// TIA Portal V20 export
DATA_BLOCK "Config"   // DB67
{ DB_Accessible_From_OPC_UA := 'FALSE' }
AUTHOR : ERsystem_FA2_DH. Kim
// stored: Access Published, DBAccessibleFromOPCUA false, DBAccessibleFromWebserver false, MemoryReserve 100, Namespace Unit1.Em3
   VAR RETAIN
      em { ExternalWritable := 'False'} : "LAF_typeEmConfiguration";
      axis { ExternalAccessible := 'False'; ExternalVisible := 'False'; ExternalWritable := 'False'} : Array[1.._.U1EM3_NO_OF_AXES] of DB_ANY;
      cam : Array[1.._.U1EM3_NO_OF_CAM] of DB_ANY;
      cmSafetyPinIdlePositionSensor { S7_SetPoint := 'True'} : "LBC_typeDigitalSignalConfiguration";
      cmRotationSafetyPinPositionSensor { S7_SetPoint := 'True'} : "LBC_typeDigitalSignalConfiguration";
      cmIonizerTopMaintDetection { S7_SetPoint := 'True'} : "LBC_typeDigitalSignalConfiguration";
      cmIonizerTopErrorDetection { S7_SetPoint := 'True'} : "LBC_typeDigitalSignalConfiguration";
      cmIonizerBtmMaintDetection { S7_SetPoint := 'True'} : "LBC_typeDigitalSignalConfiguration";
      cmIonizerBtmErrorDetection { S7_SetPoint := 'True'} : "LBC_typeDigitalSignalConfiguration";
      cmDancerEncoder { ExternalAccessible := 'False'; ExternalVisible := 'False'; ExternalWritable := 'False'} : "LBC_typeAnalogInputConfiguration";
      cmDancerElectroPneumaticRegulator { ExternalAccessible := 'False'; ExternalVisible := 'False'; ExternalWritable := 'False'} : "LBC_typeAnalogOutputConfiguration";
      cmCompensatorAxisX { ExternalAccessible := 'False'; ExternalVisible := 'False'; ExternalWritable := 'False'} : "LBC_typeAxis64PosConfiguration";
      cmMasterVirtualAxis { S7_SetPoint := 'True'} : "LBC_typeAxis64PosConfiguration";
      cmUnwinderVirtualAxis : "LBC_typeAxis64PosConfiguration";
      cmDancerFwdBwd { ExternalAccessible := 'False'; ExternalVisible := 'False'; ExternalWritable := 'False'} : "LBC_typeTwoWayActuatorConfiguration";
      cmSepaUnwinderIonizerTop { ExternalAccessible := 'False'; ExternalVisible := 'False'; ExternalWritable := 'False'; S7_SetPoint := 'True'} : "LBC_typeTwoWayActuatorConfiguration";
      cmSepaUnwinderIonizerBottom { ExternalAccessible := 'False'; ExternalVisible := 'False'; ExternalWritable := 'False'; S7_SetPoint := 'True'} : "LBC_typeTwoWayActuatorConfiguration";
      cmEpcPivot { ExternalAccessible := 'False'; ExternalVisible := 'False'; ExternalWritable := 'False'} : "LER_typeCON600Configuration";
      cmLoadCellControllerInterface { ExternalAccessible := 'False'; ExternalVisible := 'False'; ExternalWritable := 'False'} : "LBC_typeAnalogInputConfiguration";
      softCam : Struct
         cmCompensatorAxisX : "LER_typeSoftCamInterface";
         cmMasterVirtualAxis { S7_SetPoint := 'True'} : "LER_typeSoftCamInterface";
         cmUnwinderVirtualAxis { S7_SetPoint := 'True'} : "LER_typeSoftCamInterface";
      END_STRUCT;
   END_VAR
BEGIN
   em.referenceDesignator.parent := WSTRING#'U1';
   em.referenceDesignator.relative := WSTRING#'EM3 WebGuide';
   em.referenceDesignator.combined := WSTRING#'U1.EM3 WebGuide';
   axis[1] := 85;   // BA030AZSDR3_CompensatorAxisX
   axis[2] := 117;   // BA030A_MasterAxis
   axis[3] := 143;   // BA030A_UnwinderVirtualAxis
   cam[1] := 69;   // BA030AZSDR3_CompensatorAxisX_Cam
   cam[2] := 73;   // BA030AZSDR4_SepaFeedingRollerAxisB_Cam
   cmSafetyPinIdlePositionSensor.referenceDesignator := WSTRING#'DigitalSignal';
   cmSafetyPinIdlePositionSensor.onDelay := T#0MS;
   cmSafetyPinIdlePositionSensor.offDelay := T#0MS;
   cmSafetyPinIdlePositionSensor.default := FALSE;
   cmSafetyPinIdlePositionSensor.invertProcessValue := FALSE;
   cmSafetyPinIdlePositionSensor.disableAlarms := FALSE;
   cmRotationSafetyPinPositionSensor.referenceDesignator := WSTRING#'DigitalSignal';
   cmRotationSafetyPinPositionSensor.onDelay := T#0MS;
   cmRotationSafetyPinPositionSensor.offDelay := T#0MS;
   cmRotationSafetyPinPositionSensor.default := FALSE;
   cmRotationSafetyPinPositionSensor.invertProcessValue := FALSE;
   cmRotationSafetyPinPositionSensor.disableAlarms := FALSE;
   cmIonizerTopMaintDetection.referenceDesignator := WSTRING#'DigitalSignal';
   cmIonizerTopMaintDetection.onDelay := T#0MS;
   cmIonizerTopMaintDetection.offDelay := T#0MS;
   cmIonizerTopMaintDetection.default := FALSE;
   cmIonizerTopMaintDetection.invertProcessValue := FALSE;
   cmIonizerTopMaintDetection.disableAlarms := FALSE;
   cmIonizerTopErrorDetection.referenceDesignator := WSTRING#'DigitalSignal';
   cmIonizerTopErrorDetection.onDelay := T#0MS;
   cmIonizerTopErrorDetection.offDelay := T#0MS;
   cmIonizerTopErrorDetection.default := FALSE;
   cmIonizerTopErrorDetection.invertProcessValue := FALSE;
   cmIonizerTopErrorDetection.disableAlarms := FALSE;
   cmIonizerBtmMaintDetection.referenceDesignator := WSTRING#'DigitalSignal';
   cmIonizerBtmMaintDetection.onDelay := T#0MS;
   cmIonizerBtmMaintDetection.offDelay := T#0MS;
   cmIonizerBtmMaintDetection.default := FALSE;
   cmIonizerBtmMaintDetection.invertProcessValue := FALSE;
   cmIonizerBtmMaintDetection.disableAlarms := FALSE;
   cmIonizerBtmErrorDetection.referenceDesignator := WSTRING#'DigitalSignal';
   cmIonizerBtmErrorDetection.onDelay := T#0MS;
   cmIonizerBtmErrorDetection.offDelay := T#0MS;
   cmIonizerBtmErrorDetection.default := FALSE;
   cmIonizerBtmErrorDetection.invertProcessValue := FALSE;
   cmIonizerBtmErrorDetection.disableAlarms := FALSE;
   cmDancerEncoder.referenceDesignator := WSTRING#'cmDancerEncoder';
   cmDancerEncoder.physicalUnit := 'unit';
   cmDancerEncoder.isUnipolarSignal := TRUE;
   cmDancerEncoder.default := 0.0;
   cmDancerEncoder.limitHigh2 := 20.0;
   cmDancerEncoder.limitHigh1 := 15.0;
   cmDancerEncoder.limitLow1 := -15.0;
   cmDancerEncoder.limitLow2 := -50.0;
   cmDancerEncoder.processValueMax := 43.0;
   cmDancerEncoder.processValueMin := -43.0;
   cmDancerEncoder.scaleAnalogUppPoint := 27648.0;
   cmDancerEncoder.scaleAnalogLowPoint := 0.0;
   cmDancerEncoder.scaleProcessUppPoint := 43.0;
   cmDancerEncoder.scaleProcessLowPoint := -43.0;
   cmDancerEncoder.disableAlarms := FALSE;
   cmDancerElectroPneumaticRegulator.referenceDesignator := WSTRING#'cmDancerRegulator';
   cmDancerElectroPneumaticRegulator.physicalUnit := 'unit';
   cmDancerElectroPneumaticRegulator.isUnipolarSignal := TRUE;
   cmDancerElectroPneumaticRegulator.default := 0;
   cmDancerElectroPneumaticRegulator.limitHigh2 := 0.5;
   cmDancerElectroPneumaticRegulator.limitHigh1 := 0.5;
   cmDancerElectroPneumaticRegulator.limitLow1 := 0.0;
   cmDancerElectroPneumaticRegulator.limitLow2 := 0.0;
   cmDancerElectroPneumaticRegulator.processValueMax := 0.5;
   cmDancerElectroPneumaticRegulator.processValueMin := 0.0;
   cmDancerElectroPneumaticRegulator.scaleProcessUppPoint := 0.5;
   cmDancerElectroPneumaticRegulator.scaleProcessLowPoint := 0.0;
   cmDancerElectroPneumaticRegulator.scaleAnalogUppPoint := 27648.0;
   cmDancerElectroPneumaticRegulator.scaleAnalogLowPoint := 0.0;
   cmDancerElectroPneumaticRegulator.disableAlarms := TRUE;
   cmCompensatorAxisX.referenceDesignator := WSTRING#'cmCompensatorAxisX';
   cmCompensatorAxisX.disableAlarms := FALSE;
   cmCompensatorAxisX.masterControlPopUp := TRUE;
   cmCompensatorAxisX.setPositions[0].position := 0.0;
   cmCompensatorAxisX.setPositions[1].position := 50.0;
   cmCompensatorAxisX.setPositions[2].position := 70.0;
   cmCompensatorAxisX.setPositions[3..15].position := 0.0;
   cmCompensatorAxisX.setPositions[0].velocity := -1.0;
   cmCompensatorAxisX.setPositions[1..2].velocity := 30.0;
   cmCompensatorAxisX.setPositions[3..15].velocity := -1.0;
   cmCompensatorAxisX.setPositions[0].acceleration := -1.0;
   cmCompensatorAxisX.setPositions[1..2].acceleration := 30.0;
   cmCompensatorAxisX.setPositions[3..15].acceleration := -1.0;
   cmCompensatorAxisX.setPositions[0].deceleration := -1.0;
   cmCompensatorAxisX.setPositions[1..2].deceleration := 30.0;
   cmCompensatorAxisX.setPositions[3..15].deceleration := -1.0;
   cmCompensatorAxisX.setPositions[0..15]."name" := '';
   cmUnwinderVirtualAxis.referenceDesignator := WSTRING#'Axis64Pos';
   cmUnwinderVirtualAxis.disableAlarms := TRUE;
   cmUnwinderVirtualAxis.masterControlPopUp := TRUE;
   cmUnwinderVirtualAxis.setPositions[0..15].position := 0.0;
   cmUnwinderVirtualAxis.setPositions[0..15].velocity := -1.0;
   cmUnwinderVirtualAxis.setPositions[0..15].acceleration := -1.0;
   cmUnwinderVirtualAxis.setPositions[0..15].deceleration := -1.0;
   cmUnwinderVirtualAxis.setPositions[0..15]."name" := '';
   cmDancerFwdBwd.referenceDesignator := WSTRING#'cmDancerFwdBwd';
   cmDancerFwdBwd.monitoringLeavingFeedback := T#1S;
   cmDancerFwdBwd.monitoringReachingFeedback := T#1S;
   cmDancerFwdBwd.monitoringDiscrepancy := T#0MS;
   cmDancerFwdBwd.setOutputHomeContinuously := TRUE;
   cmDancerFwdBwd.setOutputWorkContinuously := TRUE;
   cmDancerFwdBwd.disableHomeCommand := FALSE;
   cmDancerFwdBwd.disableFeedbackHomePos := TRUE;
   cmDancerFwdBwd.disableFeedbackWorkPos := TRUE;
   cmDancerFwdBwd.disableAlarms := TRUE;
   cmDancerFwdBwd.resetOutputsOnError := FALSE;
   cmDancerFwdBwd.allwaysWaitOnReachingTime := FALSE;
   cmSepaUnwinderIonizerTop.referenceDesignator := WSTRING#'cmSepaUnwinderIonizerTop';
   cmSepaUnwinderIonizerTop.monitoringLeavingFeedback := T#500ms;
   cmSepaUnwinderIonizerTop.monitoringReachingFeedback := T#500ms;
   cmSepaUnwinderIonizerTop.monitoringDiscrepancy := T#0MS;
   cmSepaUnwinderIonizerTop.setOutputHomeContinuously := TRUE;
   cmSepaUnwinderIonizerTop.setOutputWorkContinuously := TRUE;
   cmSepaUnwinderIonizerTop.disableHomeCommand := FALSE;
   cmSepaUnwinderIonizerTop.disableFeedbackHomePos := TRUE;
   cmSepaUnwinderIonizerTop.disableFeedbackWorkPos := TRUE;
   cmSepaUnwinderIonizerTop.disableAlarms := TRUE;
   cmSepaUnwinderIonizerTop.resetOutputsOnError := FALSE;
   cmSepaUnwinderIonizerTop.allwaysWaitOnReachingTime := FALSE;
   cmSepaUnwinderIonizerBottom.referenceDesignator := WSTRING#'cmSepaUnwinderIonizerBtm';
   cmSepaUnwinderIonizerBottom.monitoringLeavingFeedback := T#500ms;
   cmSepaUnwinderIonizerBottom.monitoringReachingFeedback := T#500ms;
   cmSepaUnwinderIonizerBottom.monitoringDiscrepancy := T#0MS;
   cmSepaUnwinderIonizerBottom.setOutputHomeContinuously := TRUE;
   cmSepaUnwinderIonizerBottom.setOutputWorkContinuously := TRUE;
   cmSepaUnwinderIonizerBottom.disableHomeCommand := FALSE;
   cmSepaUnwinderIonizerBottom.disableFeedbackHomePos := TRUE;
   cmSepaUnwinderIonizerBottom.disableFeedbackWorkPos := TRUE;
   cmSepaUnwinderIonizerBottom.disableAlarms := TRUE;
   cmSepaUnwinderIonizerBottom.resetOutputsOnError := FALSE;
   cmSepaUnwinderIonizerBottom.allwaysWaitOnReachingTime := FALSE;
   cmLoadCellControllerInterface.referenceDesignator := WSTRING#'cmLoadCellController';
   cmLoadCellControllerInterface.physicalUnit := 'unit';
   cmLoadCellControllerInterface.isUnipolarSignal := TRUE;
   cmLoadCellControllerInterface.default := 0.0;
   cmLoadCellControllerInterface.limitHigh2 := 90.0;
   cmLoadCellControllerInterface.limitHigh1 := 80.0;
   cmLoadCellControllerInterface.limitLow1 := -80.0;
   cmLoadCellControllerInterface.limitLow2 := -90.0;
   cmLoadCellControllerInterface.processValueMax := 100.0;
   cmLoadCellControllerInterface.processValueMin := -100.0;
   cmLoadCellControllerInterface.scaleAnalogUppPoint := 27648.0;
   cmLoadCellControllerInterface.scaleAnalogLowPoint := 0.0;
   cmLoadCellControllerInterface.scaleProcessUppPoint := 100.0;
   cmLoadCellControllerInterface.scaleProcessLowPoint := -100.0;
   cmLoadCellControllerInterface.disableAlarms := TRUE;
END_DATA_BLOCK
